// TIA Portal V17 export
// export: Created 2025-03-07T09:17:46.1015387Z, ExportSetting WithDefaults, DisplayName Totally Integrated Automation Portal, DisplayVersion V17 Update 8, DisplayName TIA Portal Openness, DisplayVersion V17 Update 8, DisplayName TIA Portal Version Control Interface, DisplayVersion V17, DisplayName SINAMICS Startdrive Advanced, DisplayVersion V17 SP2, DisplayName SINAMICS Startdrive G110M, G120, G120C, G120D, G120P, G115D, DisplayVersion V17 SP2, DisplayName SINAMICS Startdrive G130, G150, S120, S150, SINAMICS MV, S210, DisplayVersion V17 SP2, DisplayName STEP 7 Professional, DisplayVersion V17 Update 8, DisplayName SINUMERIK ONE STEP 7 Toolbox, DisplayVersion V17 Update 12, DisplayName SINUMERIK 840D sl STEP 7 Toolbox, DisplayVersion V17 Update 12, DisplayName STEP 7 Safety, DisplayVersion V17 Update 6, DisplayName WinCC Advanced, DisplayVersion V17 Update 8
FUNCTION_BLOCK "FB2123_PANEL_BUTTON"   // FB2123, LAD
{ S7_Optimized_Access := 'FALSE' }
AUTHOR : ETXETAR
VERSION : 1.0
// stored: AutoNumber false, IsIECCheckEnabled false, SetENOAutomatically false, UDAEnableTagReadback false
   VAR_INPUT
      OPTIONS_0 : Byte := 2#0000_0000;   // OPTIONS 0
      START_CYCLE : Bool;   // START CYCLE / INPUT START CYCLE
      STOP_END_CYCLE : Bool;   // STOP END OF CYCLE / INPUT STOP END CYCLE
      IMMEDIATE_STOP : Bool;   // INMEDIATE STOP / INPUT IMMEDIATE STOP
      EMERGENCY_STOP : Bool;   // EMERGENCY STOP / INPUT EMERGENCY STOP
      HOME_POSITION : Bool;   // INPUT HOME POSITION
      RESET_FAULT : Bool;   // RESET FAULT / INPUT RESET FAULT
      AUTO_SELECTOR : Bool;   // INPUT SELECTOR AUTO SELECTED
      MANUAL_LOAD_SELECTOR : Bool;   // INPUT SELECTOR MANUAL LOAD SELECTED
      LOCK_UNLOCK_GATES : Bool;   // LOCK UNLOCK GATES / INPUT LOCK UNLOCK GATES
      DOOR_LAMP_COND : Bool;   // INPUT DOOR LAMP CONDITIONS
      BHG_BYPASS_GATES : Bool;   // BY PASSED SAFETY GATES MAIN PANEL / INPUT BHG BYPASS GATES
      UNLOAD_PARTS : Bool;   // INPUT UNLOAD FIXTURE PARTS
      UNLOAD_PARTS_FIXT_COND : Bool;   // INPUT UNLOAD PARTS FIXTURE CONDITIONS
      LOAD_PARTS : Bool;   // INPUT LOAD FIXTURE PARTS
      LOAD_PARTS_FIXT_COND : Bool;   // INPUT LOAD PARTS FIXTURE CONDITIONS
   END_VAR
   VAR_OUTPUT
      START_CYCLE_LAMP : Bool;   // START CYCLE LAMP
      END_OF_CYCLE_LAMP : Bool;   // END OF CYCLE LAMP
      HOME_LAMP : Bool;   // HOME POSITION LAMP
      RESET_LAMP : Bool;   // RESET LAMP
      LOCK_DOOR_LAMP : Bool;   // LOCK DOOR LAMP
      UNLOAD_LAMP : Bool;   // UNLOAD PARTS LAMP
      LOAD_LAMP : Bool;   // LOAD PARTS LAMP
      EMERGENCY_STOP_ALARM : Bool;   // EMERGENCY STOP FAULT / EMERGENCY STOP ALARM
   END_VAR
   VAR DB_SPECIFIC
      MANUAL_REQUEST : Bool;   // MANUAL REQUEST
      SEMI_REQUEST : Bool;   // SEMI REQUEST
      AUTO_REQUEST : Bool;   // AUTO REQUEST
      SETUP_REQUEST : Bool;   // SETUP REQUEST
      PARTS_UNLOADED : Bool;   // PARTS UNLOADED
      PARTS_LOADED : Bool;   // PARTS LOADED
      END_OF_CYCLE_ALARM : Bool;   // END OF CYCLE ALARM
      IMMEDIATE_STOP_ALARM : Bool;   // IMMEDIATE STOP ALARM
      HOME_POSITION_ALARM : Bool;   // HOME POSITION ALARM
      SEOC_BY_OPERATOR : Bool;   // STOP END OF CYCLE BY OPERATOR / SEOC BY OPERATOR
      MANUAL_LOADING_SEL_BUTTO : Bool;   // MANUAL LOADING SELECTOR BUTTON / MANUAL LOADING SEL BUTTO
      WARNING_GONE : Bool;   // WARNING GONE
      E_RETURN_PULSE : Bool;   // EMERGENCY RETURN PULSE
      AUX1 : Bool;   // AUX1
      AUX2 : Bool;   // AUX2
      AUX3 : Bool;   // AUX3
      AUX4 : Bool;   // AUX4
      CONDITION_HELP : Bool;   // CONDITION HELP
   END_VAR
   VAR_TEMP
      INPUTS_MASK : Byte;   // INPUT MASK
      O_BYTE_0 : Struct   // OPTIONS BYTE 0
         CHANGE_MODE_WO_PANEL_ACTIVE : Bool;   // CHANGE MODE WITHOUT PANEL ACTIVE OPTION
         MAGAZINE_PANEL : Bool;   // MAGAZINE PANEL OPTION
         PHD_PANEL : Bool;   // PART HANDLING DEVICE PANEL OPTION
         BIMANUAL_PANEL : Bool;   // SPARE OPTION
         SPARE_4 : Bool;   // SPARE OPTION
         SPARE_5 : Bool;   // SPARE OPTION
         SPARE_6 : Bool;   // SPARE OPTION
         SPARE_7 : Bool;   // SPARE OPTION
      END_STRUCT;
      DB_NUMBER : DInt;   // DB NUMBER FOR ALARM AND HELP DECODING
   END_VAR
   VAR_TEMP   // added for the SCL form of the ladder/FBD networks
      _w1 : Bool;
      _w2 : Bool;
      _w3 : Bool;
   END_VAR
BEGIN

NETWORK
TITLE = READ INSTANCE DB
      L     DINO;
      +     10#800000;
      T     #DB_NUMBER;


REGION Network 2: OPTIONS
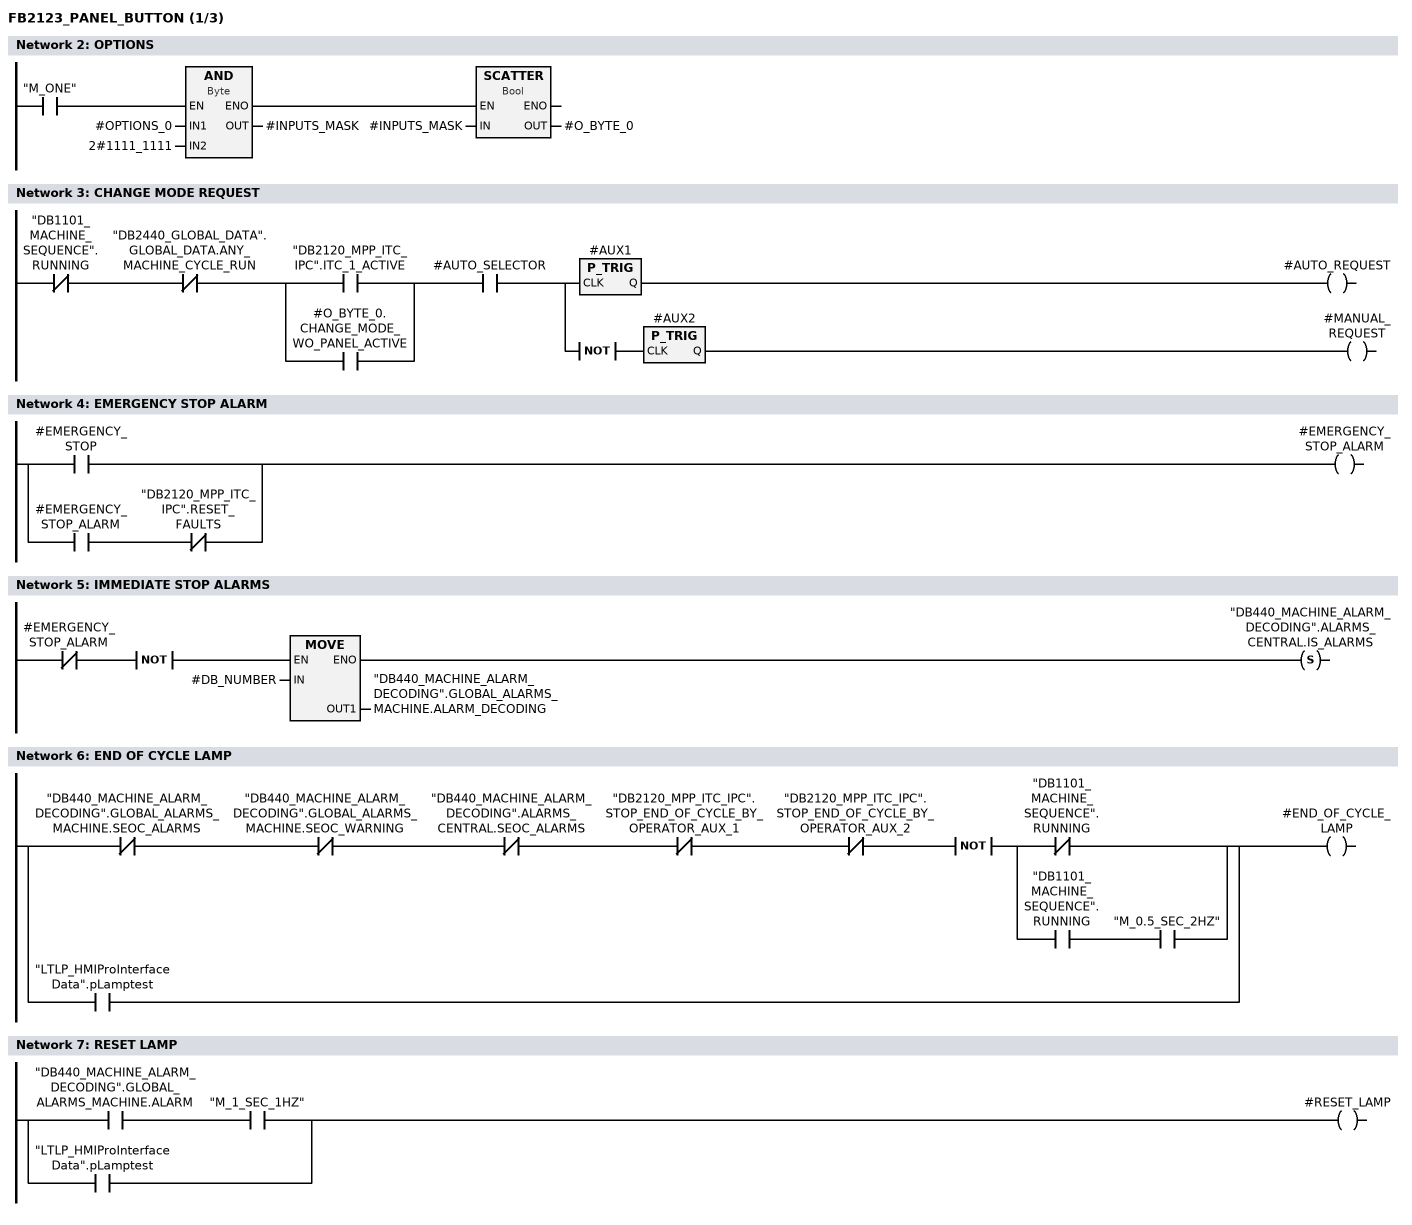
   RUNG wire#powerrail
      Contact( "M_ONE" )
      { S7_Templates := "SrcType := Byte"; S7_GenerateENO := "TRUE" } And(in1 := #OPTIONS_0, in2 := 2#1111_1111, out => #INPUTS_MASK)
      { S7_Templates := "[dest_type := Bool, src_type := Byte]" } SCATTER(IN := #INPUTS_MASK, OUT => #O_BYTE_0)
   END_RUNG
   // the same network as SCL:
   IF "M_ONE" THEN
       #INPUTS_MASK := #OPTIONS_0 AND 2#1111_1111;
       SCATTER(IN := #INPUTS_MASK, OUT => #O_BYTE_0);
   END_IF;
END_REGION

REGION Network 3: CHANGE MODE REQUEST
   RUNG wire#powerrail
      I_Contact( "DB1101_MACHINE_SEQUENCE".RUNNING )
      I_Contact( "DB2440_GLOBAL_DATA".GLOBAL_DATA.ANY_MACHINE_CYCLE_RUN )
      wire#w1
      Contact( "DB2120_MPP_ITC_IPC".ITC_1_ACTIVE )
      wire#w2
      Contact( #AUTO_SELECTOR )
      wire#w3
      P_Trig( #AUX1 )
      Coil( #AUTO_REQUEST )
   END_RUNG
   RUNG wire#w1
      Contact( #O_BYTE_0.CHANGE_MODE_WO_PANEL_ACTIVE )
   END_RUNG wire#w2
   RUNG wire#w3
      Not()
      P_Trig( #AUX2 )
      Coil( #MANUAL_REQUEST )
   END_RUNG
   // the same network as SCL:
   #_w1 := NOT "DB1101_MACHINE_SEQUENCE".RUNNING AND NOT "DB2440_GLOBAL_DATA".GLOBAL_DATA.ANY_MACHINE_CYCLE_RUN AND ("DB2120_MPP_ITC_IPC".ITC_1_ACTIVE OR #O_BYTE_0.CHANGE_MODE_WO_PANEL_ACTIVE) AND #AUTO_SELECTOR;
   #_w2 := #_w1 AND NOT #AUX1;   // rising edge
   #AUX1 := #_w1;
   #AUTO_REQUEST := #_w2;
   #_w3 := NOT #_w1 AND NOT #AUX2;   // rising edge
   #AUX2 := NOT #_w1;
   #MANUAL_REQUEST := #_w3;
END_REGION

REGION Network 4: EMERGENCY STOP ALARM
   RUNG wire#powerrail
      Contact( #EMERGENCY_STOP )
      wire#w1
      Coil( #EMERGENCY_STOP_ALARM )
   END_RUNG
   RUNG wire#powerrail
      Contact( #EMERGENCY_STOP_ALARM )
      I_Contact( "DB2120_MPP_ITC_IPC".RESET_FAULTS )
   END_RUNG wire#w1
   // the same network as SCL:
   #EMERGENCY_STOP_ALARM := #EMERGENCY_STOP OR (#EMERGENCY_STOP_ALARM AND NOT "DB2120_MPP_ITC_IPC".RESET_FAULTS);
END_REGION

REGION Network 5: IMMEDIATE STOP ALARMS
   RUNG wire#powerrail
      I_Contact( #EMERGENCY_STOP_ALARM )
      Not()
      { S7_GenerateENO := "TRUE" } Move(in := #DB_NUMBER, out1 => "DB440_MACHINE_ALARM_DECODING".GLOBAL_ALARMS_MACHINE.ALARM_DECODING)
      S_Coil( "DB440_MACHINE_ALARM_DECODING".ALARMS_CENTRAL.IS_ALARMS )
   END_RUNG
   // the same network as SCL:
   // ENO of a box is taken as its EN; it also drops when the box reports an error
   IF NOT (NOT #EMERGENCY_STOP_ALARM) THEN
       "DB440_MACHINE_ALARM_DECODING".GLOBAL_ALARMS_MACHINE.ALARM_DECODING := #DB_NUMBER;
       "DB440_MACHINE_ALARM_DECODING".ALARMS_CENTRAL.IS_ALARMS := TRUE;
   END_IF;
END_REGION

REGION Network 6: END OF CYCLE LAMP
   RUNG wire#powerrail
      I_Contact( "DB440_MACHINE_ALARM_DECODING".GLOBAL_ALARMS_MACHINE.SEOC_ALARMS )
      I_Contact( "DB440_MACHINE_ALARM_DECODING".GLOBAL_ALARMS_MACHINE.SEOC_WARNING )
      I_Contact( "DB440_MACHINE_ALARM_DECODING".ALARMS_CENTRAL.SEOC_ALARMS )
      I_Contact( "DB2120_MPP_ITC_IPC".STOP_END_OF_CYCLE_BY_OPERATOR_AUX_1 )
      I_Contact( "DB2120_MPP_ITC_IPC".STOP_END_OF_CYCLE_BY_OPERATOR_AUX_2 )
      Not()
      wire#w1
      I_Contact( "DB1101_MACHINE_SEQUENCE".RUNNING )
      wire#w2
      Coil( #END_OF_CYCLE_LAMP )
   END_RUNG
   RUNG wire#w1
      Contact( "DB1101_MACHINE_SEQUENCE".RUNNING )
      Contact( "M_0.5_SEC_2HZ" )
   END_RUNG wire#w2
   RUNG wire#powerrail
      Contact( "LTLP_HMIProInterfaceData".pLamptest )
   END_RUNG wire#w2
   // the same network as SCL:
   #END_OF_CYCLE_LAMP := (NOT (NOT "DB440_MACHINE_ALARM_DECODING".GLOBAL_ALARMS_MACHINE.SEOC_ALARMS AND NOT "DB440_MACHINE_ALARM_DECODING".GLOBAL_ALARMS_MACHINE.SEOC_WARNING AND NOT "DB440_MACHINE_ALARM_DECODING".ALARMS_CENTRAL.SEOC_ALARMS AND NOT "DB2120_MPP_ITC_IPC".STOP_END_OF_CYCLE_BY_OPERATOR_AUX_1 AND NOT "DB2120_MPP_ITC_IPC".STOP_END_OF_CYCLE_BY_OPERATOR_AUX_2) AND (NOT "DB1101_MACHINE_SEQUENCE".RUNNING OR ("DB1101_MACHINE_SEQUENCE".RUNNING AND "M_0.5_SEC_2HZ"))) OR "LTLP_HMIProInterfaceData".pLamptest;
END_REGION

REGION Network 7: RESET LAMP
   RUNG wire#powerrail
      Contact( "DB440_MACHINE_ALARM_DECODING".GLOBAL_ALARMS_MACHINE.ALARM )
      Contact( "M_1_SEC_1HZ" )
      wire#w1
      Coil( #RESET_LAMP )
   END_RUNG
   RUNG wire#powerrail
      Contact( "LTLP_HMIProInterfaceData".pLamptest )
   END_RUNG wire#w1
   // the same network as SCL:
   #RESET_LAMP := ("DB440_MACHINE_ALARM_DECODING".GLOBAL_ALARMS_MACHINE.ALARM AND "M_1_SEC_1HZ") OR "LTLP_HMIProInterfaceData".pLamptest;
END_REGION

REGION Network 8: START CYCLE LAMP
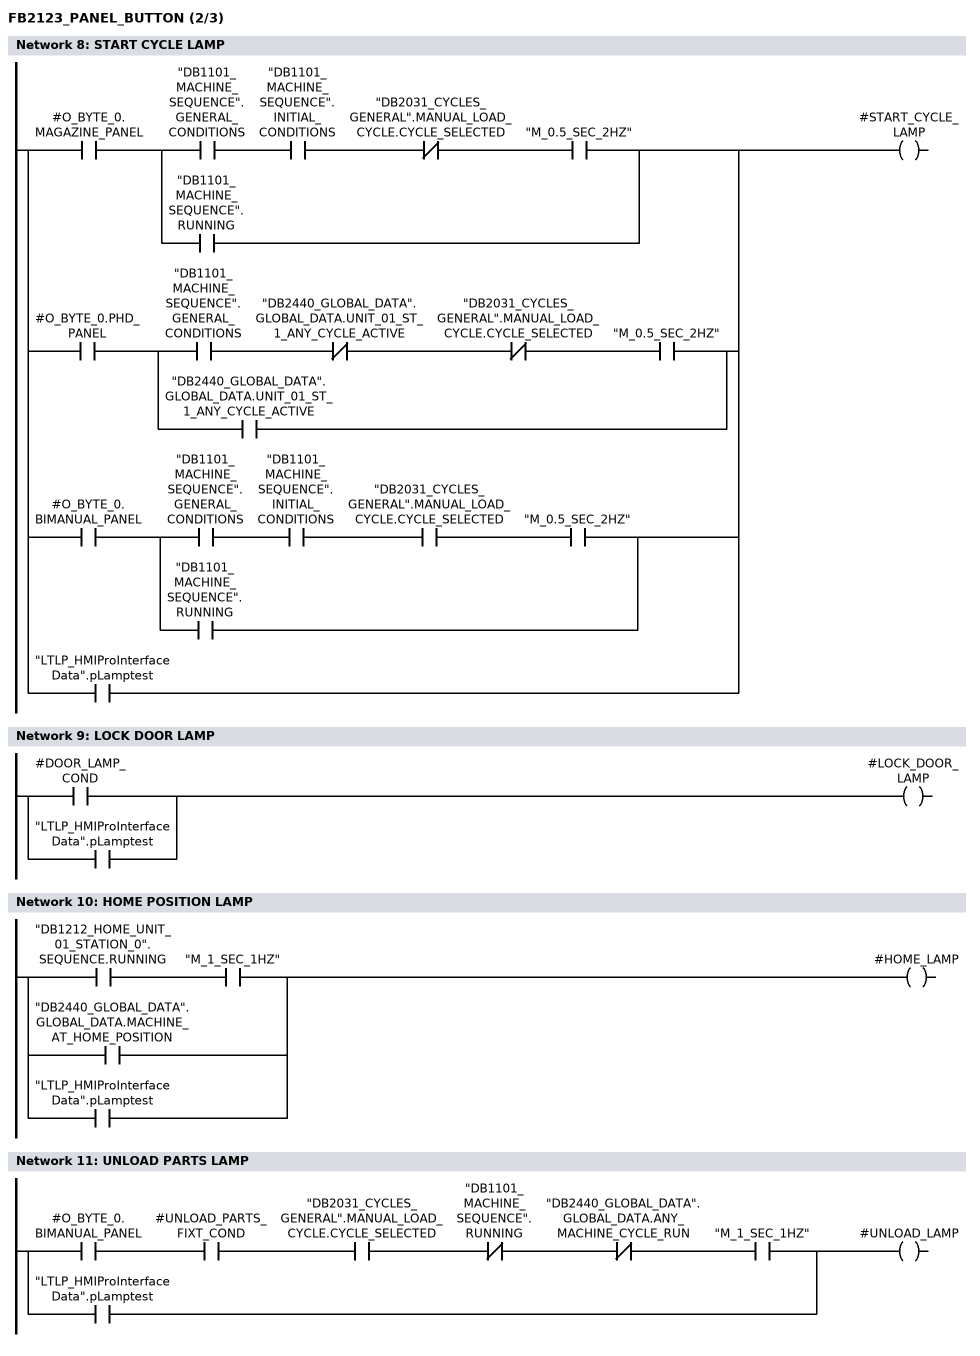
   RUNG wire#powerrail
      Contact( #O_BYTE_0.MAGAZINE_PANEL )
      wire#w1
      Contact( "DB1101_MACHINE_SEQUENCE".GENERAL_CONDITIONS )
      Contact( "DB1101_MACHINE_SEQUENCE".INITIAL_CONDITIONS )
      I_Contact( "DB2031_CYCLES_GENERAL".MANUAL_LOAD_CYCLE.CYCLE_SELECTED )
      Contact( "M_0.5_SEC_2HZ" )
      wire#w2
      Coil( #START_CYCLE_LAMP )
   END_RUNG
   RUNG wire#w1
      Contact( "DB1101_MACHINE_SEQUENCE".RUNNING )
   END_RUNG wire#w2
   RUNG wire#powerrail
      Contact( #O_BYTE_0.PHD_PANEL )
      wire#w3
      Contact( "DB1101_MACHINE_SEQUENCE".GENERAL_CONDITIONS )
      I_Contact( "DB2440_GLOBAL_DATA".GLOBAL_DATA.UNIT_01_ST_1_ANY_CYCLE_ACTIVE )
      I_Contact( "DB2031_CYCLES_GENERAL".MANUAL_LOAD_CYCLE.CYCLE_SELECTED )
      Contact( "M_0.5_SEC_2HZ" )
   END_RUNG wire#w2
   RUNG wire#w3
      Contact( "DB2440_GLOBAL_DATA".GLOBAL_DATA.UNIT_01_ST_1_ANY_CYCLE_ACTIVE )
   END_RUNG wire#w2
   RUNG wire#powerrail
      Contact( #O_BYTE_0.BIMANUAL_PANEL )
      wire#w4
      Contact( "DB1101_MACHINE_SEQUENCE".GENERAL_CONDITIONS )
      Contact( "DB1101_MACHINE_SEQUENCE".INITIAL_CONDITIONS )
      Contact( "DB2031_CYCLES_GENERAL".MANUAL_LOAD_CYCLE.CYCLE_SELECTED )
      Contact( "M_0.5_SEC_2HZ" )
   END_RUNG wire#w2
   RUNG wire#w4
      Contact( "DB1101_MACHINE_SEQUENCE".RUNNING )
   END_RUNG wire#w2
   RUNG wire#powerrail
      Contact( "LTLP_HMIProInterfaceData".pLamptest )
   END_RUNG wire#w2
   // the same network as SCL:
   #START_CYCLE_LAMP := (#O_BYTE_0.MAGAZINE_PANEL AND (("DB1101_MACHINE_SEQUENCE".GENERAL_CONDITIONS AND "DB1101_MACHINE_SEQUENCE".INITIAL_CONDITIONS AND NOT "DB2031_CYCLES_GENERAL".MANUAL_LOAD_CYCLE.CYCLE_SELECTED AND "M_0.5_SEC_2HZ") OR "DB1101_MACHINE_SEQUENCE".RUNNING)) OR (#O_BYTE_0.PHD_PANEL AND (("DB1101_MACHINE_SEQUENCE".GENERAL_CONDITIONS AND NOT "DB2440_GLOBAL_DATA".GLOBAL_DATA.UNIT_01_ST_1_ANY_CYCLE_ACTIVE AND NOT "DB2031_CYCLES_GENERAL".MANUAL_LOAD_CYCLE.CYCLE_SELECTED AND "M_0.5_SEC_2HZ") OR "DB2440_GLOBAL_DATA".GLOBAL_DATA.UNIT_01_ST_1_ANY_CYCLE_ACTIVE)) OR (#O_BYTE_0.BIMANUAL_PANEL AND (("DB1101_MACHINE_SEQUENCE".GENERAL_CONDITIONS AND "DB1101_MACHINE_SEQUENCE".INITIAL_CONDITIONS AND "DB2031_CYCLES_GENERAL".MANUAL_LOAD_CYCLE.CYCLE_SELECTED AND "M_0.5_SEC_2HZ") OR "DB1101_MACHINE_SEQUENCE".RUNNING)) OR "LTLP_HMIProInterfaceData".pLamptest;
END_REGION

REGION Network 9: LOCK DOOR LAMP
   RUNG wire#powerrail
      Contact( #DOOR_LAMP_COND )
      wire#w1
      Coil( #LOCK_DOOR_LAMP )
   END_RUNG
   RUNG wire#powerrail
      Contact( "LTLP_HMIProInterfaceData".pLamptest )
   END_RUNG wire#w1
   // the same network as SCL:
   #LOCK_DOOR_LAMP := #DOOR_LAMP_COND OR "LTLP_HMIProInterfaceData".pLamptest;
END_REGION

REGION Network 10: HOME POSITION LAMP
   RUNG wire#powerrail
      Contact( "DB1212_HOME_UNIT_01_STATION_0".SEQUENCE.RUNNING )
      Contact( "M_1_SEC_1HZ" )
      wire#w1
      Coil( #HOME_LAMP )
   END_RUNG
   RUNG wire#powerrail
      Contact( "DB2440_GLOBAL_DATA".GLOBAL_DATA.MACHINE_AT_HOME_POSITION )
   END_RUNG wire#w1
   RUNG wire#powerrail
      Contact( "LTLP_HMIProInterfaceData".pLamptest )
   END_RUNG wire#w1
   // the same network as SCL:
   #HOME_LAMP := ("DB1212_HOME_UNIT_01_STATION_0".SEQUENCE.RUNNING AND "M_1_SEC_1HZ") OR "DB2440_GLOBAL_DATA".GLOBAL_DATA.MACHINE_AT_HOME_POSITION OR "LTLP_HMIProInterfaceData".pLamptest;
END_REGION

REGION Network 11: UNLOAD PARTS LAMP
   RUNG wire#powerrail
      Contact( #O_BYTE_0.BIMANUAL_PANEL )
      Contact( #UNLOAD_PARTS_FIXT_COND )
      Contact( "DB2031_CYCLES_GENERAL".MANUAL_LOAD_CYCLE.CYCLE_SELECTED )
      I_Contact( "DB1101_MACHINE_SEQUENCE".RUNNING )
      I_Contact( "DB2440_GLOBAL_DATA".GLOBAL_DATA.ANY_MACHINE_CYCLE_RUN )
      Contact( "M_1_SEC_1HZ" )
      wire#w1
      Coil( #UNLOAD_LAMP )
   END_RUNG
   RUNG wire#powerrail
      Contact( "LTLP_HMIProInterfaceData".pLamptest )
   END_RUNG wire#w1
   // the same network as SCL:
   #UNLOAD_LAMP := (#O_BYTE_0.BIMANUAL_PANEL AND #UNLOAD_PARTS_FIXT_COND AND "DB2031_CYCLES_GENERAL".MANUAL_LOAD_CYCLE.CYCLE_SELECTED AND NOT "DB1101_MACHINE_SEQUENCE".RUNNING AND NOT "DB2440_GLOBAL_DATA".GLOBAL_DATA.ANY_MACHINE_CYCLE_RUN AND "M_1_SEC_1HZ") OR "LTLP_HMIProInterfaceData".pLamptest;
END_REGION

REGION Network 12: LOAD PARTS LAMP
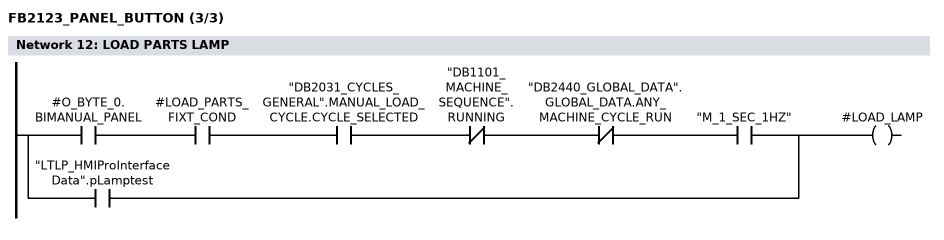
   RUNG wire#powerrail
      Contact( #O_BYTE_0.BIMANUAL_PANEL )
      Contact( #LOAD_PARTS_FIXT_COND )
      Contact( "DB2031_CYCLES_GENERAL".MANUAL_LOAD_CYCLE.CYCLE_SELECTED )
      I_Contact( "DB1101_MACHINE_SEQUENCE".RUNNING )
      I_Contact( "DB2440_GLOBAL_DATA".GLOBAL_DATA.ANY_MACHINE_CYCLE_RUN )
      Contact( "M_1_SEC_1HZ" )
      wire#w1
      Coil( #LOAD_LAMP )
   END_RUNG
   RUNG wire#powerrail
      Contact( "LTLP_HMIProInterfaceData".pLamptest )
   END_RUNG wire#w1
   // the same network as SCL:
   #LOAD_LAMP := (#O_BYTE_0.BIMANUAL_PANEL AND #LOAD_PARTS_FIXT_COND AND "DB2031_CYCLES_GENERAL".MANUAL_LOAD_CYCLE.CYCLE_SELECTED AND NOT "DB1101_MACHINE_SEQUENCE".RUNNING AND NOT "DB2440_GLOBAL_DATA".GLOBAL_DATA.ANY_MACHINE_CYCLE_RUN AND "M_1_SEC_1HZ") OR "LTLP_HMIProInterfaceData".pLamptest;
END_REGION
END_FUNCTION_BLOCK
